% RSLogix 500 project BASE.RSS, saved by version 8.10.00.18 %
PROJECT "BASE"    % processor: MicroLogix 1200 %

PROGRAM FILES
  LAD 2   3 rungs

DATA FILES
  O0 OUTPUT  4 elements
  I1 INPUT  4 elements
  S2 STATUS  66 elements
  B3 BINARY  1 elements
  T4 TIMER  1 elements
  C5 COUNTER  1 elements
  R6 CONTROL  1 elements
  N7 INTEGER  1 elements
  F8 FLOAT  1 elements

LADDER 2
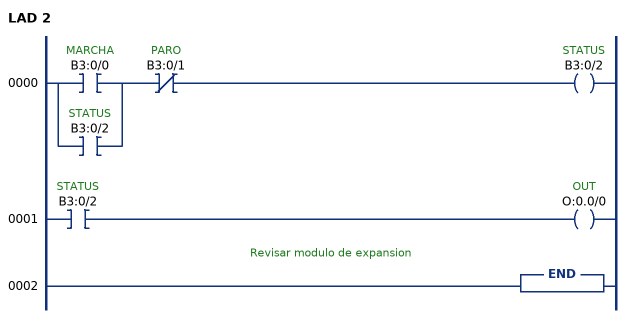
% Rung: 0 %
SOR BST XIC B3:0/0 NXB XIC B3:0/2 BND XIO B3:0/1 OTE B3:0/2 EOR
%   B3:0/0  MARCHA %
%   B3:0/2  STATUS %
%   B3:0/1  PARO %
% Rung: 1 %
SOR XIC B3:0/2 OTE O:0.0/0 EOR
%   B3:0/2  STATUS %
%   O:0.0/0  OUT %
% Rung: 2 %
% Revisar modulo de expansion %
SOR END EOR

REVISION NOTES
  0: Cambio de IP
